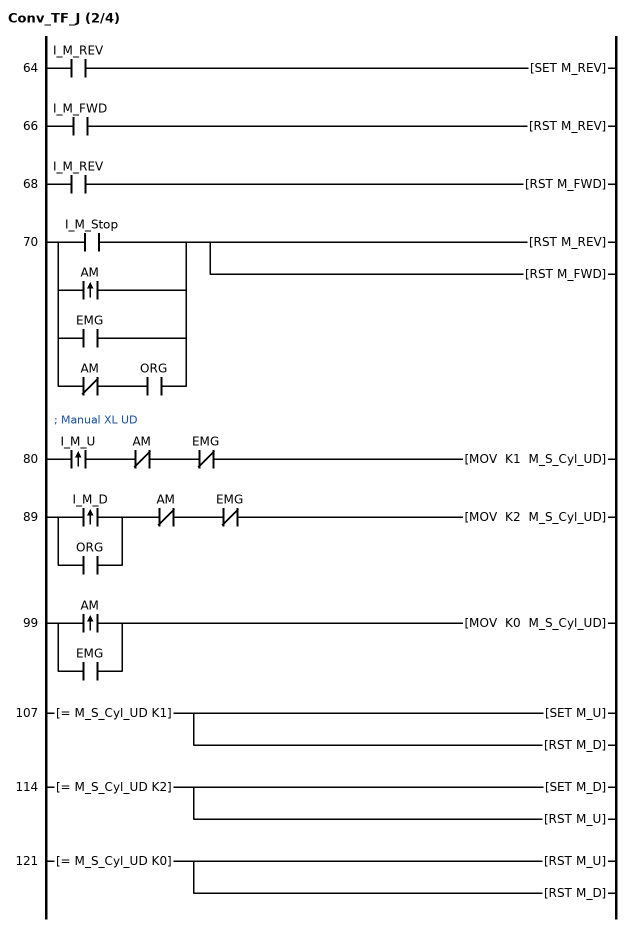
[picture p24: ladder of Conv_TF_J, rungs at steps 64 to 121]
64    LD      I_M_REV
      SET     M_REV
66    LD      I_M_FWD
      RST     M_REV
68    LD      I_M_REV
      RST     M_FWD
70    LD      I_M_Stop
      ORP     AM
      OR      EMG
      LDI     AM
      AND     ORG
      ORB
      RST     M_REV
      RST     M_FWD
; Manual XL UD
80    LDP     I_M_U
      ANI     AM
      ANI     EMG
      MOV     K1 M_S_Cyl_UD
89    LDP     I_M_D
      OR      ORG
      ANI     AM
      ANI     EMG
      MOV     K2 M_S_Cyl_UD
99    LDP     AM
      OR      EMG
      MOV     K0 M_S_Cyl_UD
107   LD=     M_S_Cyl_UD K1
      SET     M_U
      RST     M_D
114   LD=     M_S_Cyl_UD K2
      SET     M_D
      RST     M_U
121   LD=     M_S_Cyl_UD K0
      RST     M_U
      RST     M_D
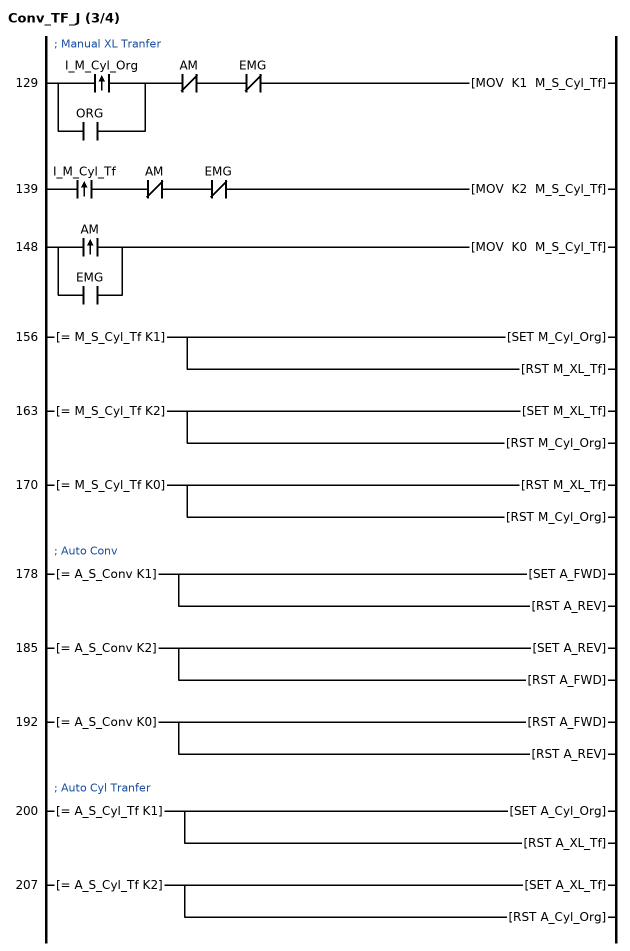
; Manual XL Tranfer
129   LDP     I_M_Cyl_Org
      OR      ORG
      ANI     AM
      ANI     EMG
      MOV     K1 M_S_Cyl_Tf
139   LDP     I_M_Cyl_Tf
      ANI     AM
      ANI     EMG
      MOV     K2 M_S_Cyl_Tf
148   LDP     AM
      OR      EMG
      MOV     K0 M_S_Cyl_Tf
156   LD=     M_S_Cyl_Tf K1
      SET     M_Cyl_Org
      RST     M_XL_Tf
163   LD=     M_S_Cyl_Tf K2
      SET     M_XL_Tf
      RST     M_Cyl_Org
170   LD=     M_S_Cyl_Tf K0
      RST     M_XL_Tf
      RST     M_Cyl_Org
; Auto Conv
178   LD=     A_S_Conv K1
      SET     A_FWD
      RST     A_REV
185   LD=     A_S_Conv K2
      SET     A_REV
      RST     A_FWD
192   LD=     A_S_Conv K0
      RST     A_FWD
      RST     A_REV
; Auto Cyl Tranfer
200   LD=     A_S_Cyl_Tf K1
      SET     A_Cyl_Org
      RST     A_XL_Tf
207   LD=     A_S_Cyl_Tf K2
      SET     A_XL_Tf
      RST     A_Cyl_Org
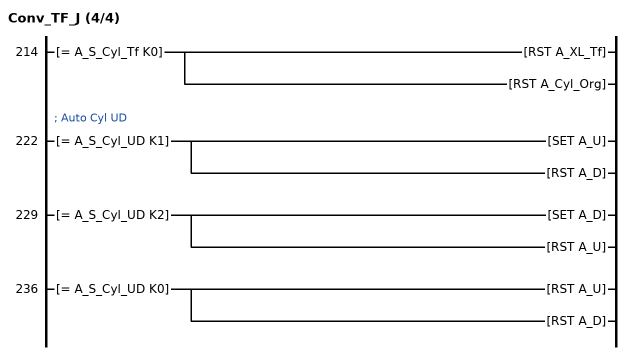
214   LD=     A_S_Cyl_Tf K0
      RST     A_XL_Tf
      RST     A_Cyl_Org
; Auto Cyl UD
222   LD=     A_S_Cyl_UD K1
      SET     A_U
      RST     A_D
229   LD=     A_S_Cyl_UD K2
      SET     A_D
      RST     A_U
236   LD=     A_S_Cyl_UD K0
      RST     A_U
      RST     A_D
END_FUNCTION_BLOCK

FUNCTION_BLOCK Conv_Wait
VAR_INPUT
  AM : BOOL;
  EMG : BOOL;
END_VAR
VAR_OUTPUT
  FWD : BOOL;
  Stopper_Up : BOOL;
  Stopper_Down : BOOL;
END_VAR
VAR
  M_FWD : BOOL;
  M_U : BOOL;
  A_U : BOOL;
  M_D : BOOL;
  A_D : BOOL;
  M_S_Stp : INT;
END_VAR
VAR_INPUT
  I_M_FWD : BOOL;
  I_M_Stop : BOOL;
  I_M_U : BOOL;
  I_M_D : BOOL;
  A_FWD : BOOL;
  A_S_Stp : INT;
  L_C : BOOL;
  ORG : BOOL;
END_VAR
VAR_OUTPUT
  S_Org : BOOL;
END_VAR
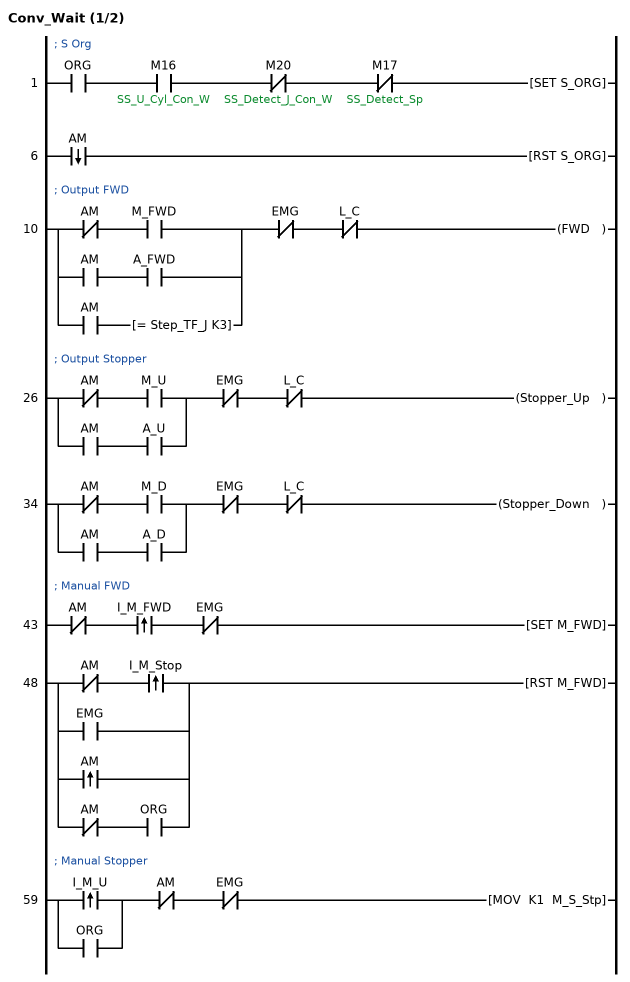
; S Org
1     LD      ORG
      AND     M16  ; SS_U_Cyl_Con_W
      ANI     M20  ; SS_Detect_J_Con_W
      ANI     M17  ; SS_Detect_Sp
      SET     S_ORG
6     LDF     AM
      RST     S_ORG
; Output FWD
10    LDI     AM
      AND     M_FWD
      LD      AM
      AND     A_FWD
      ORB
      LD      AM
      AND=    Step_TF_J K3
      ORB
      ANI     EMG
      ANI     L_C
      OUT     FWD
; Output Stopper
26    LDI     AM
      AND     M_U
      LD      AM
      AND     A_U
      ORB
      ANI     EMG
      ANI     L_C
      OUT     Stopper_Up
34    LDI     AM
      AND     M_D
      LD      AM
      AND     A_D
      ORB
      ANI     EMG
      ANI     L_C
      OUT     Stopper_Down
; Manual FWD
43    LDI     AM
      ANDP    I_M_FWD
      ANI     EMG
      SET     M_FWD
48    LDI     AM
      ANDP    I_M_Stop
      OR      EMG
      ORP     AM
      LDI     AM
      AND     ORG
      ORB
      RST     M_FWD
; Manual Stopper
59    LDP     I_M_U
      OR      ORG
      ANI     AM
      ANI     EMG
      MOV     K1 M_S_Stp
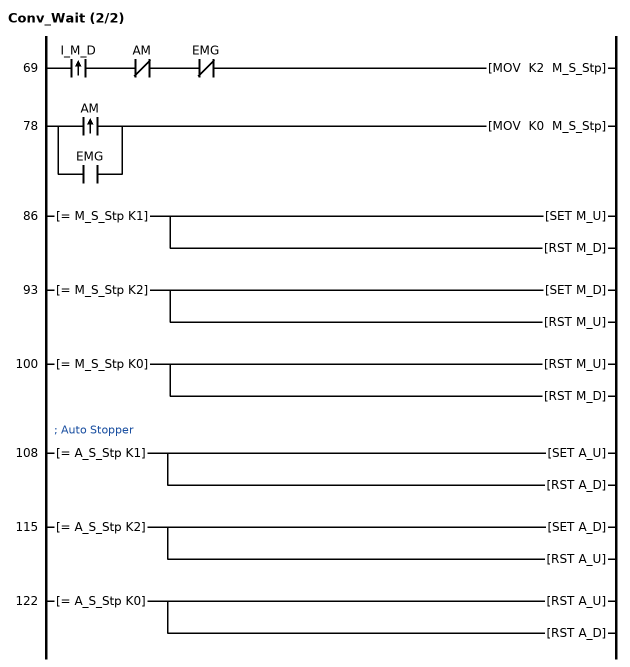
69    LDP     I_M_D
      ANI     AM
      ANI     EMG
      MOV     K2 M_S_Stp
78    LDP     AM
      OR      EMG
      MOV     K0 M_S_Stp
86    LD=     M_S_Stp K1
      SET     M_U
      RST     M_D
93    LD=     M_S_Stp K2
      SET     M_D
      RST     M_U
100   LD=     M_S_Stp K0
      RST     M_U
      RST     M_D
; Auto Stopper
108   LD=     A_S_Stp K1
      SET     A_U
      RST     A_D
115   LD=     A_S_Stp K2
      SET     A_D
      RST     A_U
122   LD=     A_S_Stp K0
      RST     A_U
      RST     A_D
END_FUNCTION_BLOCK

FUNCTION_BLOCK C_Cyl_TF_J
VAR_INPUT
  AM : BOOL;
  EMG : BOOL;
END_VAR
VAR
  M_U : BOOL;
  A_U : BOOL;
  M_D : BOOL;
  A_D : BOOL;
  M_S_Cyl_UD : INT;
  M_Org_XL_Tf : BOOL;
  A_Org_XL_Tf : BOOL;
  M_Tf_XL_Tf : BOOL;
  A_Tf_XL_Tf : BOOL;
END_VAR
VAR_INPUT
  I_M_U : BOOL;
  I_M_D : BOOL;
  I_M_Sol_Org : BOOL;
  I_M_Sol_Tf : BOOL;
  A_Status_XL_U : INT;
END_VAR
VAR
  M_Status_XL_Tf : INT;
END_VAR
VAR_INPUT
  A_S_Cyl_Tf : INT;
  ORG : BOOL;
END_VAR
VAR_OUTPUT
  XL_U : BOOL;
  XL_D : BOOL;
  Sol_Org : BOOL;
  Sol_Tranfer : BOOL;
  S_Org : BOOL;
END_VAR
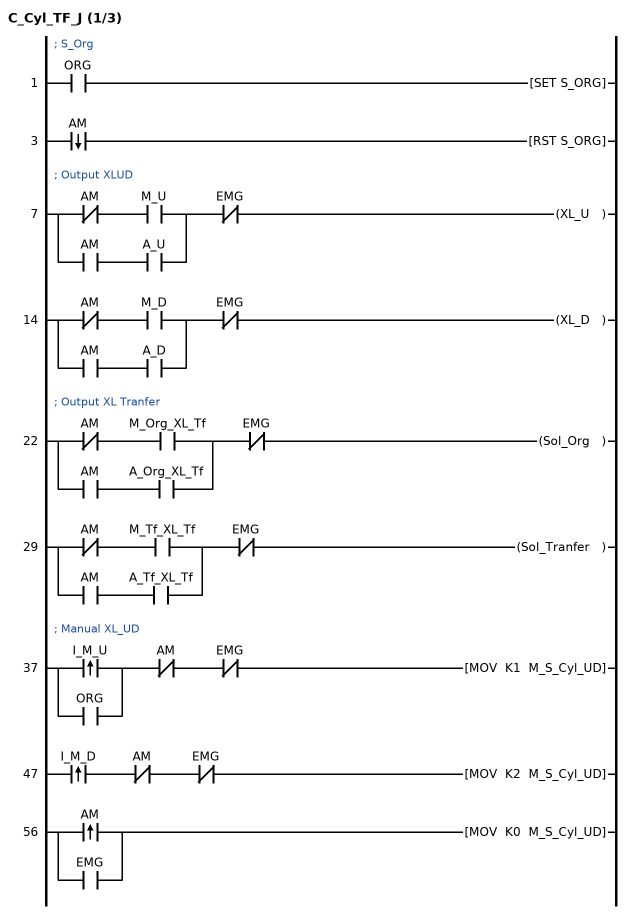
; S_Org
1     LD      ORG
      SET     S_ORG
3     LDF     AM
      RST     S_ORG
; Output XLUD
7     LDI     AM
      AND     M_U
      LD      AM
      AND     A_U
      ORB
      ANI     EMG
      OUT     XL_U
14    LDI     AM
      AND     M_D
      LD      AM
      AND     A_D
      ORB
      ANI     EMG
      OUT     XL_D
; Output XL Tranfer
22    LDI     AM
      AND     M_Org_XL_Tf
      LD      AM
      AND     A_Org_XL_Tf
      ORB
      ANI     EMG
      OUT     Sol_Org
29    LDI     AM
      AND     M_Tf_XL_Tf
      LD      AM
      AND     A_Tf_XL_Tf
      ORB
      ANI     EMG
      OUT     Sol_Tranfer
; Manual XL_UD
37    LDP     I_M_U
      OR      ORG
      ANI     AM
      ANI     EMG
      MOV     K1 M_S_Cyl_UD
47    LDP     I_M_D
      ANI     AM
      ANI     EMG
      MOV     K2 M_S_Cyl_UD
56    LDP     AM
      OR      EMG
      MOV     K0 M_S_Cyl_UD
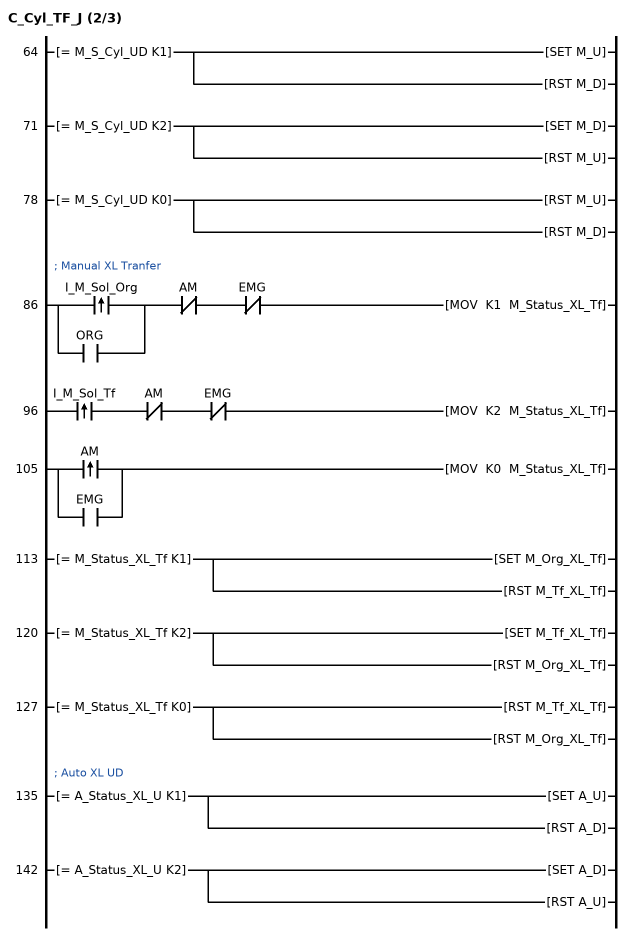
64    LD=     M_S_Cyl_UD K1
      SET     M_U
      RST     M_D
71    LD=     M_S_Cyl_UD K2
      SET     M_D
      RST     M_U
78    LD=     M_S_Cyl_UD K0
      RST     M_U
      RST     M_D
; Manual XL Tranfer
86    LDP     I_M_Sol_Org
      OR      ORG
      ANI     AM
      ANI     EMG
      MOV     K1 M_Status_XL_Tf
96    LDP     I_M_Sol_Tf
      ANI     AM
      ANI     EMG
      MOV     K2 M_Status_XL_Tf
105   LDP     AM
      OR      EMG
      MOV     K0 M_Status_XL_Tf
113   LD=     M_Status_XL_Tf K1
      SET     M_Org_XL_Tf
      RST     M_Tf_XL_Tf
120   LD=     M_Status_XL_Tf K2
      SET     M_Tf_XL_Tf
      RST     M_Org_XL_Tf
127   LD=     M_Status_XL_Tf K0
      RST     M_Tf_XL_Tf
      RST     M_Org_XL_Tf
; Auto XL UD
135   LD=     A_Status_XL_U K1
      SET     A_U
      RST     A_D
142   LD=     A_Status_XL_U K2
      SET     A_D
      RST     A_U
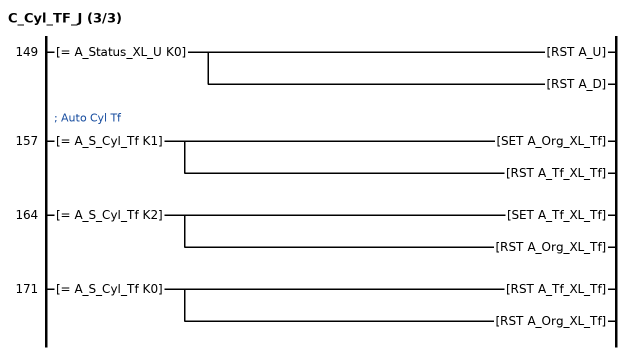
149   LD=     A_Status_XL_U K0
      RST     A_U
      RST     A_D
; Auto Cyl Tf
157   LD=     A_S_Cyl_Tf K1
      SET     A_Org_XL_Tf
      RST     A_Tf_XL_Tf
164   LD=     A_S_Cyl_Tf K2
      SET     A_Tf_XL_Tf
      RST     A_Org_XL_Tf
171   LD=     A_S_Cyl_Tf K0
      RST     A_Tf_XL_Tf
      RST     A_Org_XL_Tf
END_FUNCTION_BLOCK

FUNCTION_BLOCK C_Cyl_TF_SP
VAR_INPUT
  AM : BOOL;
  EMG : BOOL;
  I_M_U : BOOL;
  I_M_D : BOOL;
  I_M_Sol_Org : BOOL;
  I_M_Sol_Tf : BOOL;
  I_M_XL_Kep_SP1 : BOOL;
  I_M_XL_Nha_SP1 : BOOL;
END_VAR
VAR
  Step_Run : INT;
  Flag_Run : BOOL;
  Full_XL_Ready : BOOL;
  Delay_Kep_Sp : TIMER;
END_VAR
VAR_INPUT
  I_M_XL_Kep_SP2 : BOOL;
  I_M_XL_Nha_SP2 : BOOL;
  A_Status_XL_U : INT;
  A_S_Cyl_Tf : INT;
  A_S_Cyl_Kep_1 : INT;
  A_S_Cyl_Kep_2 : INT;
  ORG : BOOL;
END_VAR
VAR_OUTPUT
  XL_U : BOOL;
  XL_D : BOOL;
  Sol_Org : BOOL;
  Sol_Tranfer : BOOL;
  XL_Kep_SP1 : BOOL;
  XL_Mo_SP1 : BOOL;
  XL_Kep_SP2 : BOOL;
  XL_Mo_SP2 : BOOL;
END_VAR
VAR
  M_U : BOOL;
  A_U : BOOL;
  M_D : BOOL;
  A_D : BOOL;
  M_S_Cyl_UD : INT;
  M_Org_XL_Tf : BOOL;
  A_Org_XL_Tf : BOOL;
  M_Tf_XL_Tf : BOOL;
  A_Tf_XL_Tf : BOOL;
  M_Status_XL_Tf : INT;
  M_Kep_SP1 : BOOL;
  A_Kep_SP1 : BOOL;
  M_Nha_SP1 : BOOL;
  A_Nha_SP1 : BOOL;
  M_Status_XL_Kep_Sp1 : INT;
  M_Kep_SP2 : BOOL;
  A_Kep_SP2 : BOOL;
  M_Nha_SP2 : BOOL;
  A_Nha_SP2 : BOOL;
  M_Status_XL_Kep_Sp2 : INT;
END_VAR
VAR_OUTPUT
  S_ORG : BOOL;
END_VAR
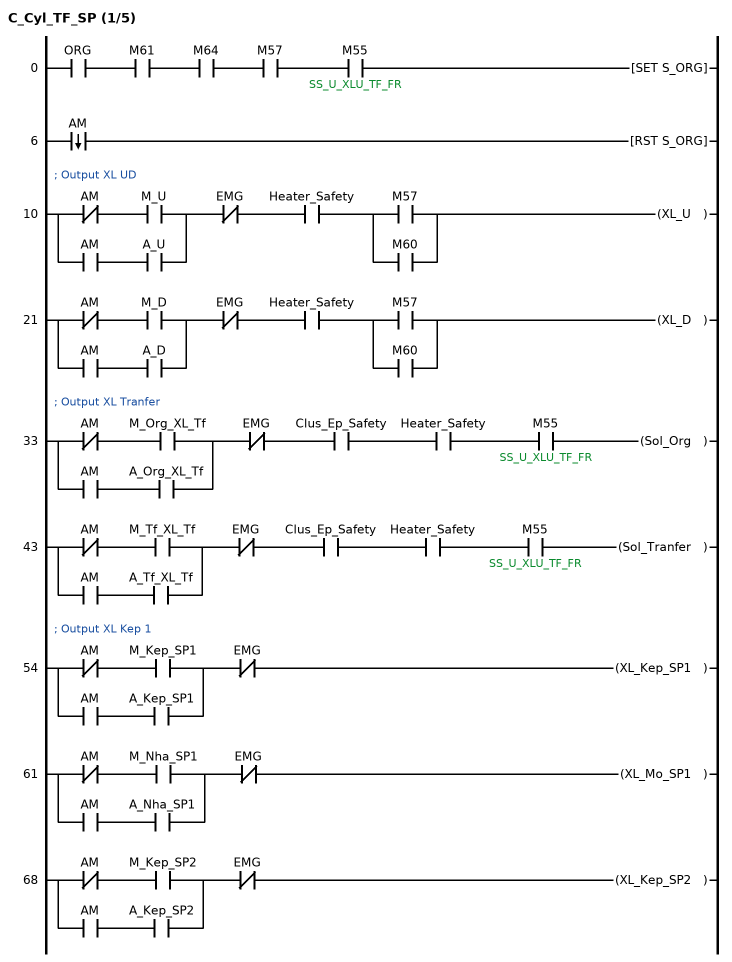
0     LD      ORG
      AND     M61
      AND     M64
      AND     M57
      AND     M55  ; SS_U_XLU_TF_FR
      SET     S_ORG
6     LDF     AM
      RST     S_ORG
; Output XL UD
10    LDI     AM
      AND     M_U
      LD      AM
      AND     A_U
      ORB
      ANI     EMG
      AND     Heater_Safety
      LD      M57
      OR      M60
      ANB
      OUT     XL_U
21    LDI     AM
      AND     M_D
      LD      AM
      AND     A_D
      ORB
      ANI     EMG
      AND     Heater_Safety
      LD      M57
      OR      M60
      ANB
      OUT     XL_D
; Output XL Tranfer
33    LDI     AM
      AND     M_Org_XL_Tf
      LD      AM
      AND     A_Org_XL_Tf
      ORB
      ANI     EMG
      AND     Clus_Ep_Safety
      AND     Heater_Safety
      AND     M55  ; SS_U_XLU_TF_FR
      OUT     Sol_Org
43    LDI     AM
      AND     M_Tf_XL_Tf
      LD      AM
      AND     A_Tf_XL_Tf
      ORB
      ANI     EMG
      AND     Clus_Ep_Safety
      AND     Heater_Safety
      AND     M55  ; SS_U_XLU_TF_FR
      OUT     Sol_Tranfer
; Output XL Kep 1
54    LDI     AM
      AND     M_Kep_SP1
      LD      AM
      AND     A_Kep_SP1
      ORB
      ANI     EMG
      OUT     XL_Kep_SP1
61    LDI     AM
      AND     M_Nha_SP1
      LD      AM
      AND     A_Nha_SP1
      ORB
      ANI     EMG
      OUT     XL_Mo_SP1
68    LDI     AM
      AND     M_Kep_SP2
      LD      AM
      AND     A_Kep_SP2
      ORB
      ANI     EMG
      OUT     XL_Kep_SP2
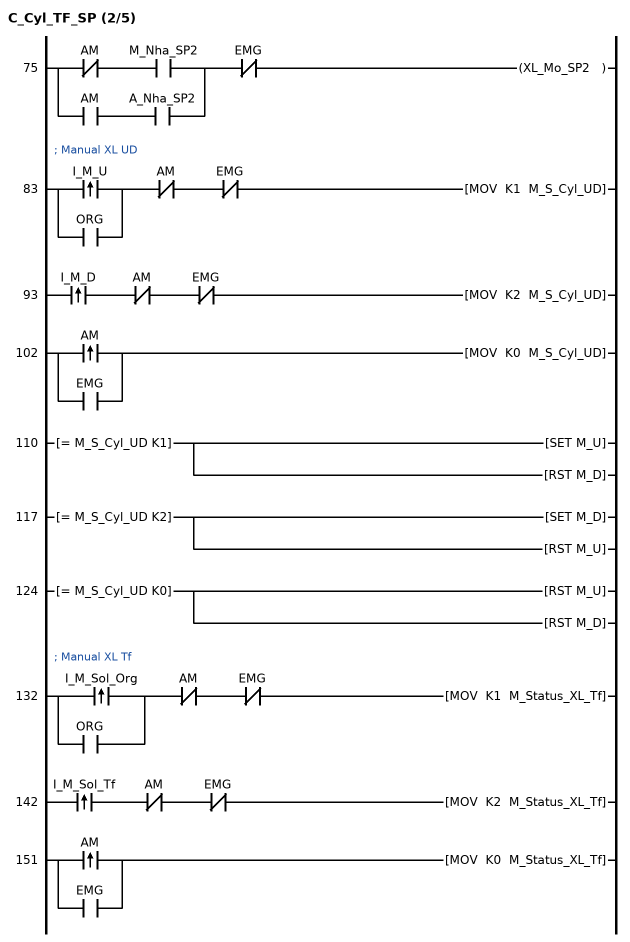
75    LDI     AM
      AND     M_Nha_SP2
      LD      AM
      AND     A_Nha_SP2
      ORB
      ANI     EMG
      OUT     XL_Mo_SP2
; Manual XL UD
83    LDP     I_M_U
      OR      ORG
      ANI     AM
      ANI     EMG
      MOV     K1 M_S_Cyl_UD
93    LDP     I_M_D
      ANI     AM
      ANI     EMG
      MOV     K2 M_S_Cyl_UD
102   LDP     AM
      OR      EMG
      MOV     K0 M_S_Cyl_UD
110   LD=     M_S_Cyl_UD K1
      SET     M_U
      RST     M_D
117   LD=     M_S_Cyl_UD K2
      SET     M_D
      RST     M_U
124   LD=     M_S_Cyl_UD K0
      RST     M_U
      RST     M_D
; Manual XL Tf
132   LDP     I_M_Sol_Org
      OR      ORG
      ANI     AM
      ANI     EMG
      MOV     K1 M_Status_XL_Tf
142   LDP     I_M_Sol_Tf
      ANI     AM
      ANI     EMG
      MOV     K2 M_Status_XL_Tf
151   LDP     AM
      OR      EMG
      MOV     K0 M_Status_XL_Tf
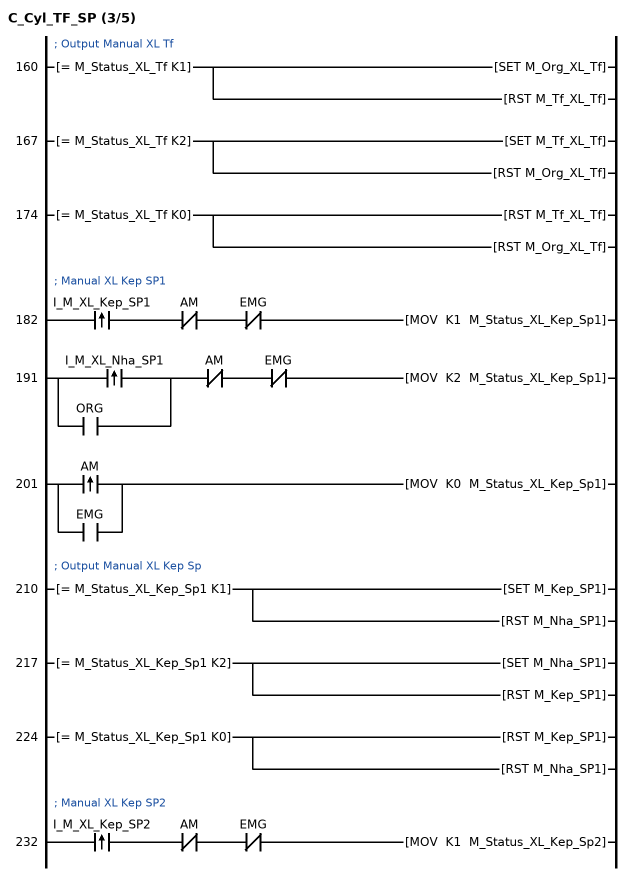
; Output Manual XL Tf
160   LD=     M_Status_XL_Tf K1
      SET     M_Org_XL_Tf
      RST     M_Tf_XL_Tf
167   LD=     M_Status_XL_Tf K2
      SET     M_Tf_XL_Tf
      RST     M_Org_XL_Tf
174   LD=     M_Status_XL_Tf K0
      RST     M_Tf_XL_Tf
      RST     M_Org_XL_Tf
; Manual XL Kep SP1
182   LDP     I_M_XL_Kep_SP1
      ANI     AM
      ANI     EMG
      MOV     K1 M_Status_XL_Kep_Sp1
191   LDP     I_M_XL_Nha_SP1
      OR      ORG
      ANI     AM
      ANI     EMG
      MOV     K2 M_Status_XL_Kep_Sp1
201   LDP     AM
      OR      EMG
      MOV     K0 M_Status_XL_Kep_Sp1
; Output Manual XL Kep Sp
210   LD=     M_Status_XL_Kep_Sp1 K1
      SET     M_Kep_SP1
      RST     M_Nha_SP1
217   LD=     M_Status_XL_Kep_Sp1 K2
      SET     M_Nha_SP1
      RST     M_Kep_SP1
224   LD=     M_Status_XL_Kep_Sp1 K0
      RST     M_Kep_SP1
      RST     M_Nha_SP1
; Manual XL Kep SP2
232   LDP     I_M_XL_Kep_SP2
      ANI     AM
      ANI     EMG
      MOV     K1 M_Status_XL_Kep_Sp2
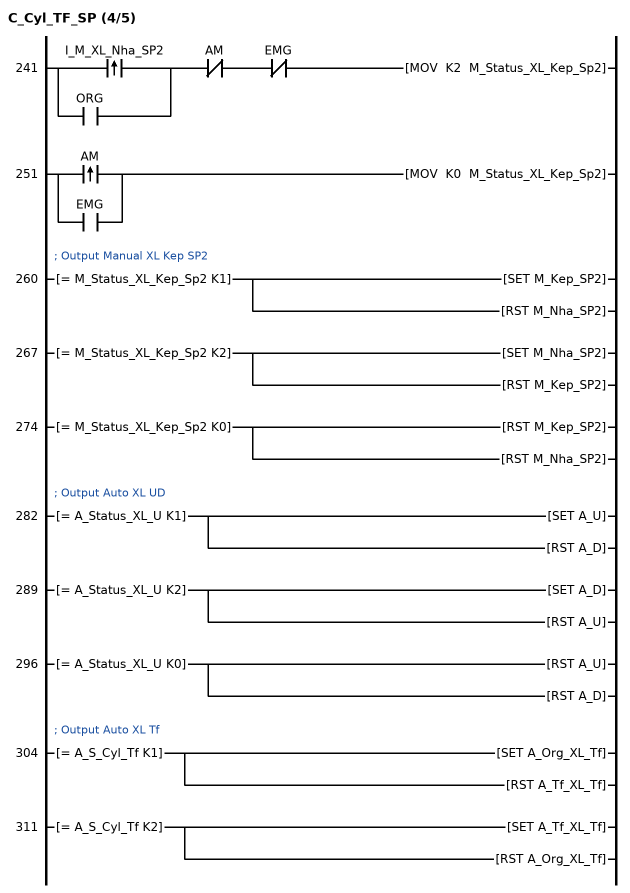
241   LDP     I_M_XL_Nha_SP2
      OR      ORG
      ANI     AM
      ANI     EMG
      MOV     K2 M_Status_XL_Kep_Sp2
251   LDP     AM
      OR      EMG
      MOV     K0 M_Status_XL_Kep_Sp2
; Output Manual XL Kep SP2
260   LD=     M_Status_XL_Kep_Sp2 K1
      SET     M_Kep_SP2
      RST     M_Nha_SP2
267   LD=     M_Status_XL_Kep_Sp2 K2
      SET     M_Nha_SP2
      RST     M_Kep_SP2
274   LD=     M_Status_XL_Kep_Sp2 K0
      RST     M_Kep_SP2
      RST     M_Nha_SP2
; Output Auto XL UD
282   LD=     A_Status_XL_U K1
      SET     A_U
      RST     A_D
289   LD=     A_Status_XL_U K2
      SET     A_D
      RST     A_U
296   LD=     A_Status_XL_U K0
      RST     A_U
      RST     A_D
; Output Auto XL Tf
304   LD=     A_S_Cyl_Tf K1
      SET     A_Org_XL_Tf
      RST     A_Tf_XL_Tf
311   LD=     A_S_Cyl_Tf K2
      SET     A_Tf_XL_Tf
      RST     A_Org_XL_Tf
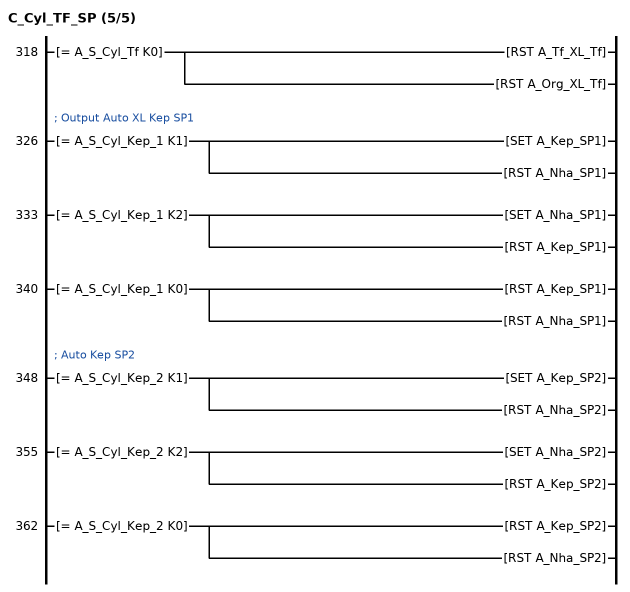
318   LD=     A_S_Cyl_Tf K0
      RST     A_Tf_XL_Tf
      RST     A_Org_XL_Tf
; Output Auto XL Kep SP1
326   LD=     A_S_Cyl_Kep_1 K1
      SET     A_Kep_SP1
      RST     A_Nha_SP1
333   LD=     A_S_Cyl_Kep_1 K2
      SET     A_Nha_SP1
      RST     A_Kep_SP1
340   LD=     A_S_Cyl_Kep_1 K0
      RST     A_Kep_SP1
      RST     A_Nha_SP1
; Auto Kep SP2
348   LD=     A_S_Cyl_Kep_2 K1
      SET     A_Kep_SP2
      RST     A_Nha_SP2
355   LD=     A_S_Cyl_Kep_2 K2
      SET     A_Nha_SP2
      RST     A_Kep_SP2
362   LD=     A_S_Cyl_Kep_2 K0
      RST     A_Kep_SP2
      RST     A_Nha_SP2
END_FUNCTION_BLOCK

FUNCTION_BLOCK Conv_Out
VAR_INPUT
  AM : BOOL;
  EMG : BOOL;
END_VAR
VAR_OUTPUT
  R_FWD : BOOL;
  Stopper_Up : BOOL;
  Stopper_Down : BOOL;
  Cyl_U_Jig : BOOL;
  Cyl_D_Jig : BOOL;
END_VAR
VAR_INPUT
  I_M_U_S : BOOL;
  I_M_D_S : BOOL;
  I_M_U_Jig : BOOL;
  I_M_D_Jig : BOOL;
  I_M_FWD : BOOL;
  I_M_Stop : BOOL;
END_VAR
VAR
  M_FWD : BOOL;
  M_U_Jig : BOOL;
  A_U_Jig : BOOL;
  M_S_Cyl_UD : INT;
  M_D_Jig : BOOL;
  A_D_Jig : BOOL;
  M_U_S : BOOL;
  A_U_S : BOOL;
  M_D_S : BOOL;
  A_D_S : BOOL;
  M_S_Stp : INT;
END_VAR
VAR_INPUT
  ORG : BOOL;
END_VAR
VAR_OUTPUT
  S_Org : BOOL;
  Sol_Do1 : BOOL;
  Sol_Do2 : BOOL;
END_VAR
VAR_INPUT
  A_S_Cyl_UD : INT;
  A_S_Stp : INT;
  A_FWD : BOOL;
  I_M_Do1 : BOOL;
  I_M_Do2 : BOOL;
  A_S_Do : INT;
END_VAR
VAR
  M_Do1 : BOOL;
  A_Do1 : BOOL;
  M_Do2 : BOOL;
  A_Do2 : BOOL;
  M_S_Do : INT;
END_VAR
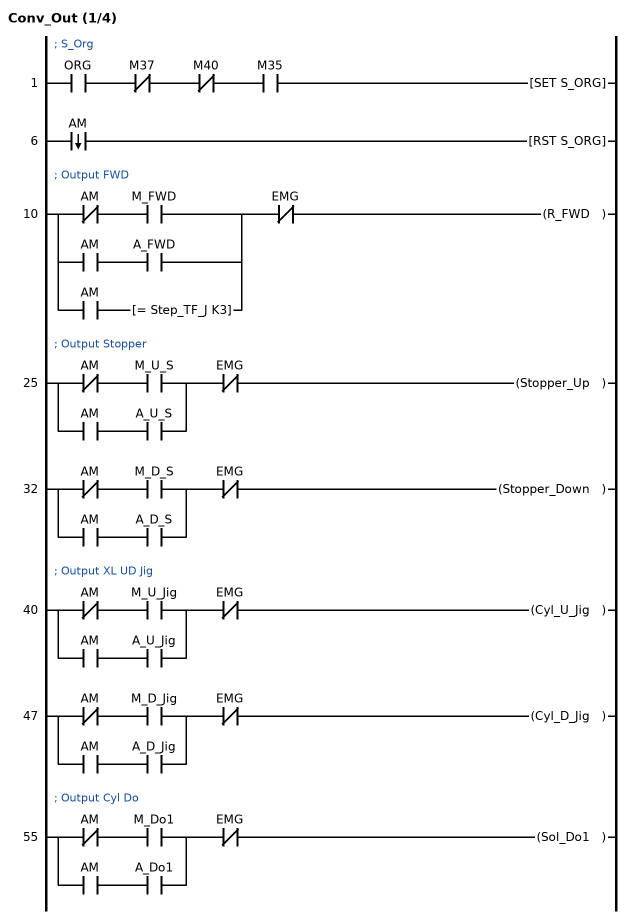
; S_Org
1     LD      ORG
      ANI     M37
      ANI     M40
      AND     M35
      SET     S_ORG
6     LDF     AM
      RST     S_ORG
; Output FWD
10    LDI     AM
      AND     M_FWD
      LD      AM
      AND     A_FWD
      ORB
      LD      AM
      AND=    Step_TF_J K3
      ORB
      ANI     EMG
      OUT     R_FWD
; Output Stopper
25    LDI     AM
      AND     M_U_S
      LD      AM
      AND     A_U_S
      ORB
      ANI     EMG
      OUT     Stopper_Up
32    LDI     AM
      AND     M_D_S
      LD      AM
      AND     A_D_S
      ORB
      ANI     EMG
      OUT     Stopper_Down
; Output XL UD Jig
40    LDI     AM
      AND     M_U_Jig
      LD      AM
      AND     A_U_Jig
      ORB
      ANI     EMG
      OUT     Cyl_U_Jig
47    LDI     AM
      AND     M_D_Jig
      LD      AM
      AND     A_D_Jig
      ORB
      ANI     EMG
      OUT     Cyl_D_Jig
; Output Cyl Do
55    LDI     AM
      AND     M_Do1
      LD      AM
      AND     A_Do1
      ORB
      ANI     EMG
      OUT     Sol_Do1
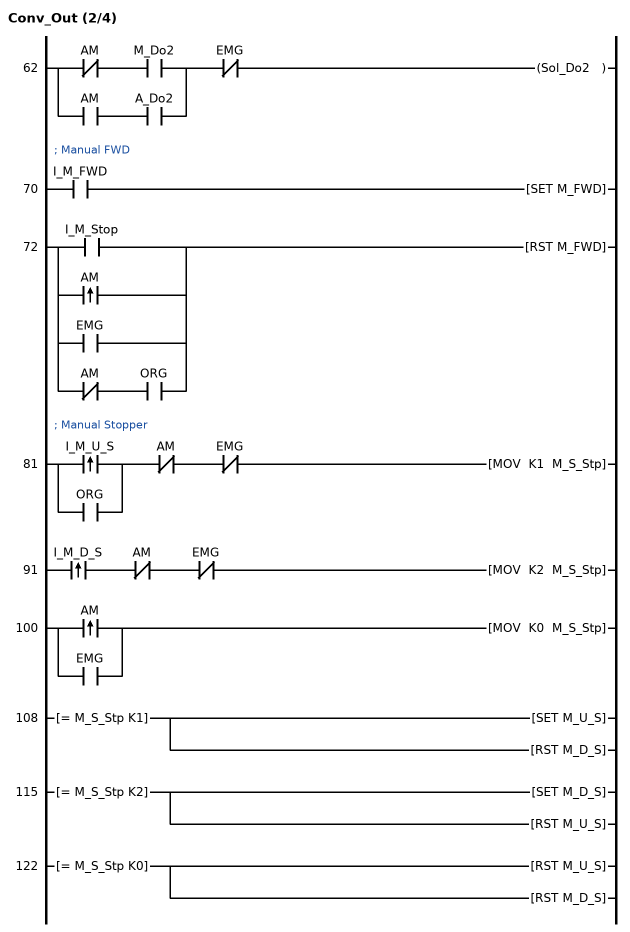
62    LDI     AM
      AND     M_Do2
      LD      AM
      AND     A_Do2
      ORB
      ANI     EMG
      OUT     Sol_Do2
; Manual FWD
70    LD      I_M_FWD
      SET     M_FWD
72    LD      I_M_Stop
      ORP     AM
      OR      EMG
      LDI     AM
      AND     ORG
      ORB
      RST     M_FWD
; Manual Stopper
81    LDP     I_M_U_S
      OR      ORG
      ANI     AM
      ANI     EMG
      MOV     K1 M_S_Stp
91    LDP     I_M_D_S
      ANI     AM
      ANI     EMG
      MOV     K2 M_S_Stp
100   LDP     AM
      OR      EMG
      MOV     K0 M_S_Stp
108   LD=     M_S_Stp K1
      SET     M_U_S
      RST     M_D_S
115   LD=     M_S_Stp K2
      SET     M_D_S
      RST     M_U_S
122   LD=     M_S_Stp K0
      RST     M_U_S
      RST     M_D_S
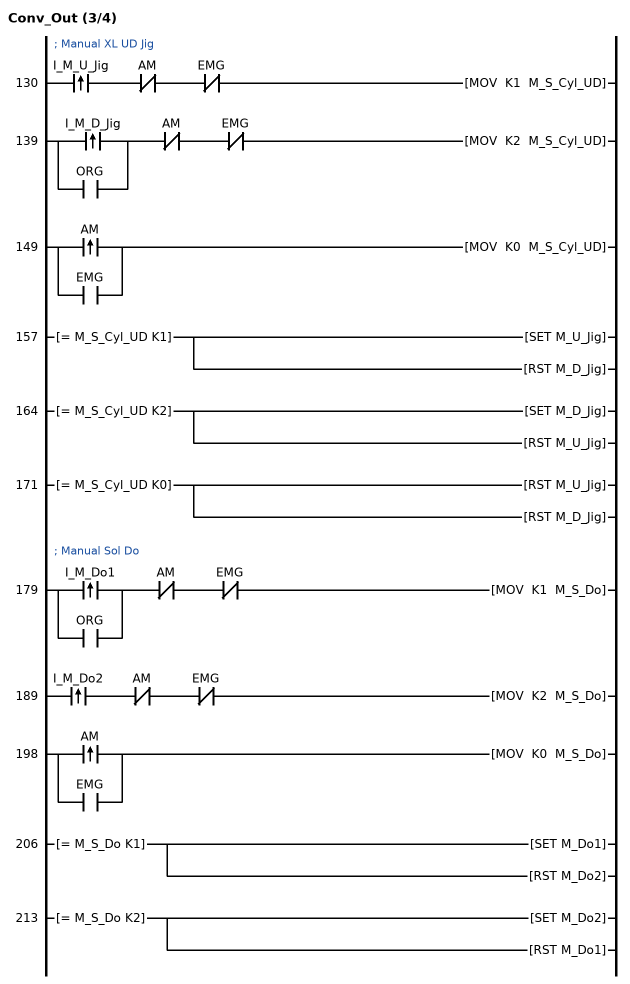
; Manual XL UD Jig
130   LDP     I_M_U_Jig
      ANI     AM
      ANI     EMG
      MOV     K1 M_S_Cyl_UD
139   LDP     I_M_D_Jig
      OR      ORG
      ANI     AM
      ANI     EMG
      MOV     K2 M_S_Cyl_UD
149   LDP     AM
      OR      EMG
      MOV     K0 M_S_Cyl_UD
157   LD=     M_S_Cyl_UD K1
      SET     M_U_Jig
      RST     M_D_Jig
164   LD=     M_S_Cyl_UD K2
      SET     M_D_Jig
      RST     M_U_Jig
171   LD=     M_S_Cyl_UD K0
      RST     M_U_Jig
      RST     M_D_Jig
; Manual Sol Do
179   LDP     I_M_Do1
      OR      ORG
      ANI     AM
      ANI     EMG
      MOV     K1 M_S_Do
189   LDP     I_M_Do2
      ANI     AM
      ANI     EMG
      MOV     K2 M_S_Do
198   LDP     AM
      OR      EMG
      MOV     K0 M_S_Do
206   LD=     M_S_Do K1
      SET     M_Do1
      RST     M_Do2
213   LD=     M_S_Do K2
      SET     M_Do2
      RST     M_Do1
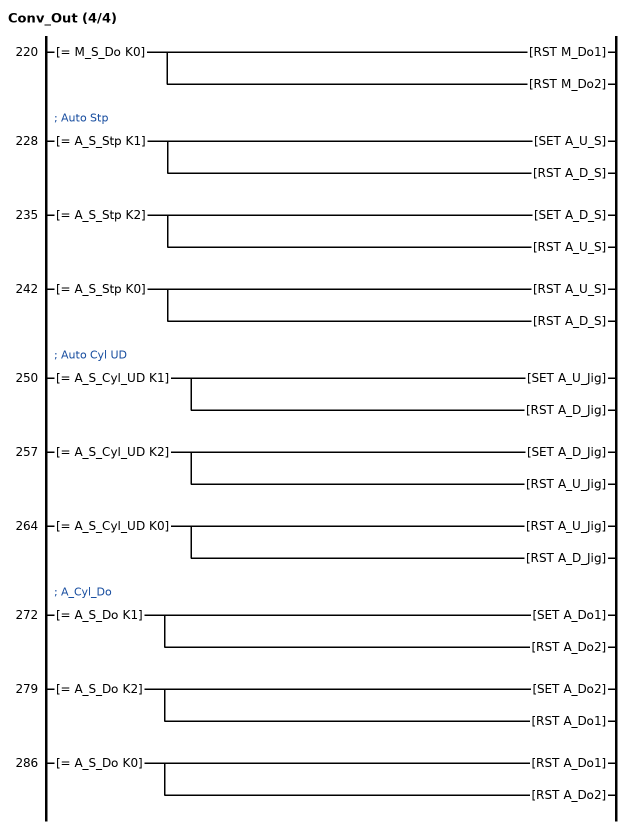
220   LD=     M_S_Do K0
      RST     M_Do1
      RST     M_Do2
; Auto Stp
228   LD=     A_S_Stp K1
      SET     A_U_S
      RST     A_D_S
235   LD=     A_S_Stp K2
      SET     A_D_S
      RST     A_U_S
242   LD=     A_S_Stp K0
      RST     A_U_S
      RST     A_D_S
; Auto Cyl UD
250   LD=     A_S_Cyl_UD K1
      SET     A_U_Jig
      RST     A_D_Jig
257   LD=     A_S_Cyl_UD K2
      SET     A_D_Jig
      RST     A_U_Jig
264   LD=     A_S_Cyl_UD K0
      RST     A_U_Jig
      RST     A_D_Jig
; A_Cyl_Do
272   LD=     A_S_Do K1
      SET     A_Do1
      RST     A_Do2
279   LD=     A_S_Do K2
      SET     A_Do2
      RST     A_Do1
286   LD=     A_S_Do K0
      RST     A_Do1
      RST     A_Do2
END_FUNCTION_BLOCK

FUNCTION_BLOCK Heater
VAR_INPUT
  AM : BOOL;
  EMG : BOOL;
END_VAR
VAR_OUTPUT
  ON_Heater : BOOL;
  XL_U : BOOL;
  XL_D : BOOL;
  ON_Center : BOOL;
  OFF_Center : BOOL;
END_VAR
VAR_INPUT
  I_M_U : BOOL;
  I_M_D : BOOL;
  I_M_On_Center : BOOL;
  I_M_Off_Center : BOOL;
END_VAR
VAR
  M_U : BOOL;
  A_U : BOOL;
  M_D : BOOL;
  A_D : BOOL;
  M_S_Cyl_UD : INT;
  M_ON_Center : BOOL;
  A_ON_Center : BOOL;
  M_OFF_Center : BOOL;
  A_OFF_Center : BOOL;
  M_Status_Center : INT;
END_VAR
VAR_INPUT
  I_ON_Heater : BOOL;
  A_ON_Heater : BOOL;
  A_S_Cyl_UD : INT;
  A_Status_Center : INT;
  T_Real : REAL;
  T_Limit : REAL;
  ORG : BOOL;
END_VAR
VAR_OUTPUT
  S_ORG : BOOL;
END_VAR
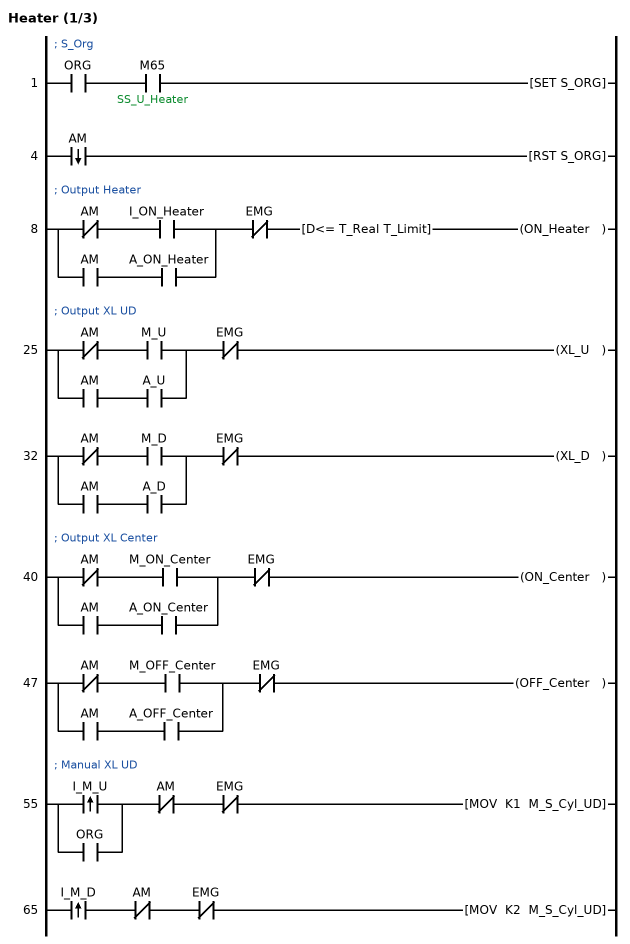
; S_Org
1     LD      ORG
      AND     M65  ; SS_U_Heater
      SET     S_ORG
4     LDF     AM
      RST     S_ORG
; Output Heater
8     LDI     AM
      AND     I_ON_Heater
      LD      AM
      AND     A_ON_Heater
      ORB
      ANI     EMG
      ANDD<=  T_Real T_Limit
      OUT     ON_Heater
; Output XL UD
25    LDI     AM
      AND     M_U
      LD      AM
      AND     A_U
      ORB
      ANI     EMG
      OUT     XL_U
32    LDI     AM
      AND     M_D
      LD      AM
      AND     A_D
      ORB
      ANI     EMG
      OUT     XL_D
; Output XL Center
40    LDI     AM
      AND     M_ON_Center
      LD      AM
      AND     A_ON_Center
      ORB
      ANI     EMG
      OUT     ON_Center
47    LDI     AM
      AND     M_OFF_Center
      LD      AM
      AND     A_OFF_Center
      ORB
      ANI     EMG
      OUT     OFF_Center
; Manual XL UD
55    LDP     I_M_U
      OR      ORG
      ANI     AM
      ANI     EMG
      MOV     K1 M_S_Cyl_UD
65    LDP     I_M_D
      ANI     AM
      ANI     EMG
      MOV     K2 M_S_Cyl_UD
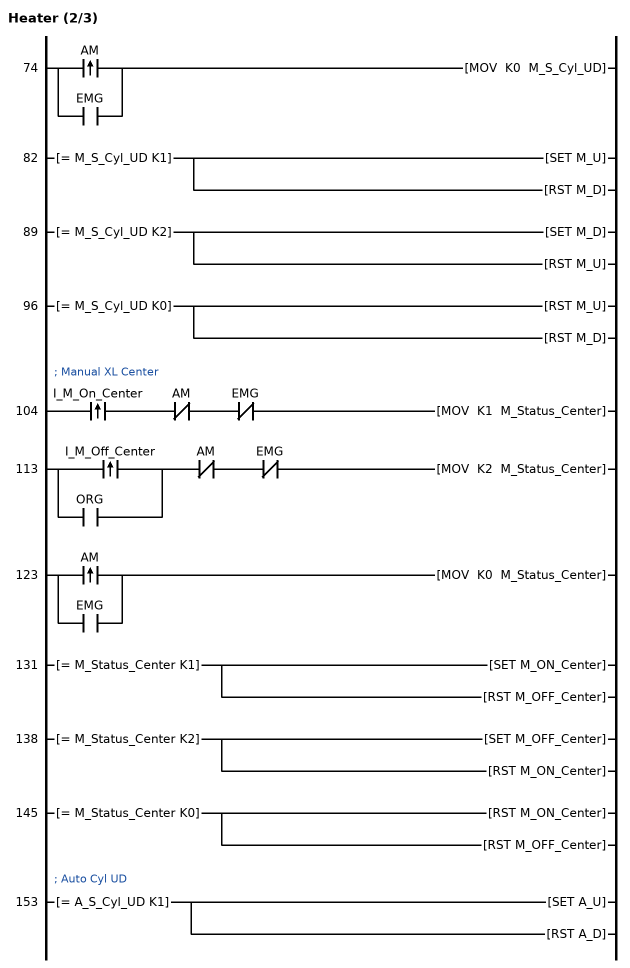
74    LDP     AM
      OR      EMG
      MOV     K0 M_S_Cyl_UD
82    LD=     M_S_Cyl_UD K1
      SET     M_U
      RST     M_D
89    LD=     M_S_Cyl_UD K2
      SET     M_D
      RST     M_U
96    LD=     M_S_Cyl_UD K0
      RST     M_U
      RST     M_D
; Manual XL Center
104   LDP     I_M_On_Center
      ANI     AM
      ANI     EMG
      MOV     K1 M_Status_Center
113   LDP     I_M_Off_Center
      OR      ORG
      ANI     AM
      ANI     EMG
      MOV     K2 M_Status_Center
123   LDP     AM
      OR      EMG
      MOV     K0 M_Status_Center
131   LD=     M_Status_Center K1
      SET     M_ON_Center
      RST     M_OFF_Center
138   LD=     M_Status_Center K2
      SET     M_OFF_Center
      RST     M_ON_Center
145   LD=     M_Status_Center K0
      RST     M_ON_Center
      RST     M_OFF_Center
; Auto Cyl UD
153   LD=     A_S_Cyl_UD K1
      SET     A_U
      RST     A_D
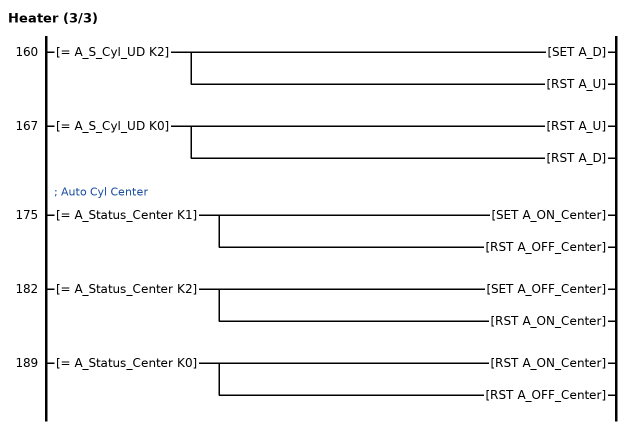
160   LD=     A_S_Cyl_UD K2
      SET     A_D
      RST     A_U
167   LD=     A_S_Cyl_UD K0
      RST     A_U
      RST     A_D
; Auto Cyl Center
175   LD=     A_Status_Center K1
      SET     A_ON_Center
      RST     A_OFF_Center
182   LD=     A_Status_Center K2
      SET     A_OFF_Center
      RST     A_ON_Center
189   LD=     A_Status_Center K0
      RST     A_ON_Center
      RST     A_OFF_Center
END_FUNCTION_BLOCK

FUNCTION_BLOCK Ctr_MC
VAR_INPUT
  I_AM : BOOL;
END_VAR
VAR_OUTPUT
  Flag_Run : BOOL;
  EMG : BOOL;
  AM : BOOL;
  R_Home : BOOL;
END_VAR
VAR_INPUT
  I_RST : BOOL;
  I_ORG : BOOL;
  I_EMG : INT;
END_VAR
VAR
  Delay_R_H : TIMER;
  T_R_H : BOOL;
  T_Auto : TIMER;
END_VAR
VAR_OUTPUT
  Red : BOOL;
  Yel : BOOL;
  Gre : BOOL;
  Buzzer : BOOL;
END_VAR
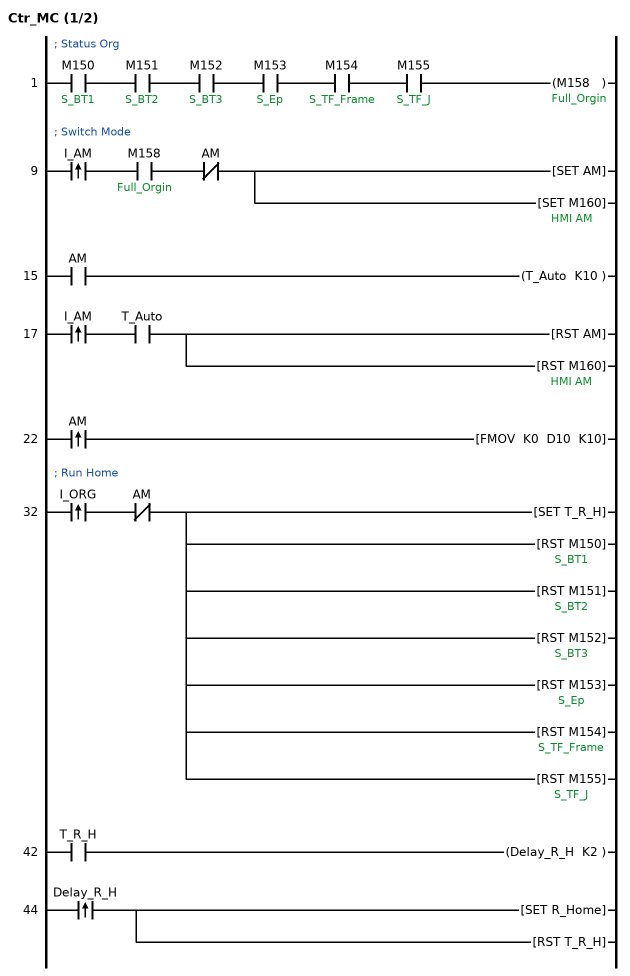
; Status Org
1     LD      M150  ; S_BT1
      AND     M151  ; S_BT2
      AND     M152  ; S_BT3
      AND     M153  ; S_Ep
      AND     M154  ; S_TF_Frame
      AND     M155  ; S_TF_J
      OUT     M158  ; Full_Orgin
; Switch Mode
9     LDP     I_AM
      AND     M158  ; Full_Orgin
      ANI     AM
      SET     AM
      SET     M160  ; HMI AM
15    LD      AM
      OUT     T_Auto K10
17    LDP     I_AM
      AND     T_Auto
      RST     AM
      RST     M160  ; HMI AM
22    LDP     AM
      FMOV    K0 D10 K10
; Run Home
32    LDP     I_ORG
      ANI     AM
      SET     T_R_H
      RST     M150  ; S_BT1
      RST     M151  ; S_BT2
      RST     M152  ; S_BT3
      RST     M153  ; S_Ep
      RST     M154  ; S_TF_Frame
      RST     M155  ; S_TF_J
42    LD      T_R_H
      OUT     Delay_R_H K2
44    LDP     Delay_R_H
      SET     R_Home
      RST     T_R_H
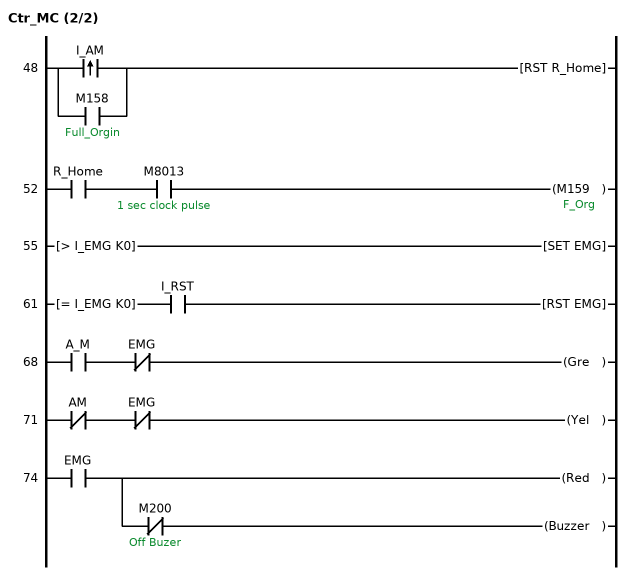
48    LDP     I_AM
      OR      M158  ; Full_Orgin
      RST     R_Home
52    LD      R_Home
      AND     M8013  ; 1 sec clock pulse
      OUT     M159  ; F_Org
55    LD>     I_EMG K0
      SET     EMG
61    LD=     I_EMG K0
      AND     I_RST
      RST     EMG
68    LD      A_M
      ANI     EMG
      OUT     Gre
71    LDI     AM
      ANI     EMG
      OUT     Yel
74    LD      EMG
      OUT     Red
      ANI     M200  ; Off Buzer
      OUT     Buzzer
END_FUNCTION_BLOCK

FUNCTION_BLOCK C_ShellCage
VAR_INPUT
  AM : BOOL;
  EMG : BOOL;
  I_M_U_DT : BOOL;
  I_M_D_DT : BOOL;
  I_M_Kep : BOOL;
  I_M_Nha : BOOL;
  I_M_Do_Org : BOOL;
  I_M_Do_Lap : BOOL;
  I_M_U_S : BOOL;
  I_M_D_S : BOOL;
  I_M_U_Jig : BOOL;
  I_M_D_Jig : BOOL;
END_VAR
VAR_OUTPUT
  U_Cyl_DT : BOOL;
  D_Cyl_DT : BOOL;
  Kep : BOOL;
  Nha : BOOL;
  Stopper_Up : BOOL;
  Stopper_Down : BOOL;
  Cyl_U_Jig : BOOL;
  Cyl_D_Jig : BOOL;
  Cyl_U_DT_J : BOOL;
  Cyl_D_DT_J : BOOL;
END_VAR
VAR
  M_U_DT : BOOL;
  A_U_DT : BOOL;
  M_D_DT : BOOL;
  A_D_DT : BOOL;
  M_S_Cyl_DT : INT;
  M_Kep : BOOL;
  A_Kep : BOOL;
  M_Nha : BOOL;
  A_Nha : BOOL;
  M_S_Cyl_Kep : INT;
  M_U_S : BOOL;
  A_U_S : BOOL;
  M_D_S : BOOL;
  A_D_S : BOOL;
  M_S_Stp : INT;
  M_U_Jig : BOOL;
  A_U_Jig : BOOL;
  M_D_Jig : BOOL;
  A_D_Jig : BOOL;
  M_S_UD_J : INT;
END_VAR
VAR_INPUT
  I_M_U_DT_Jig : BOOL;
  I_M_D_DT_Jig : BOOL;
END_VAR
VAR
  M_U_DT_J : BOOL;
  A_U_DT_J : BOOL;
  M_D_DT_J : BOOL;
  A_D_DT_J : BOOL;
  M_S_DT_J : INT;
END_VAR
VAR_INPUT
  A_S_Cyl_Kep : INT;
  A_S_Cyl_DT : INT;
  A_S_Stp : INT;
  A_S_UD_J : INT;
  A_S_DT_J : INT;
  ORG : BOOL;
END_VAR
VAR_OUTPUT
  S_Org : BOOL;
END_VAR
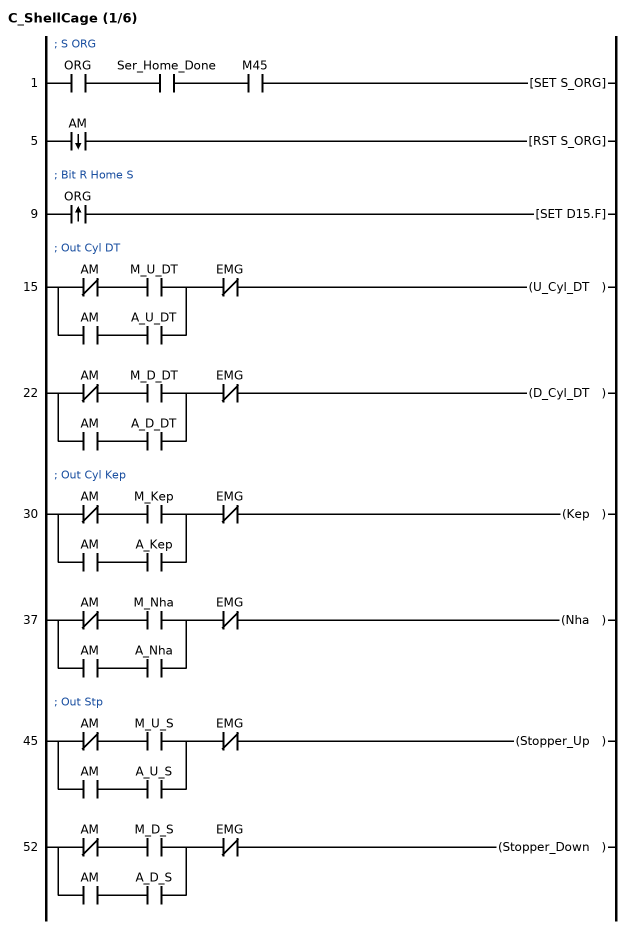
; S ORG
1     LD      ORG
      AND     Ser_Home_Done
      AND     M45
      SET     S_ORG
5     LDF     AM
      RST     S_ORG
; Bit R Home S
9     LDP     ORG
      SET     D15.F
; Out Cyl DT
15    LDI     AM
      AND     M_U_DT
      LD      AM
      AND     A_U_DT
      ORB
      ANI     EMG
      OUT     U_Cyl_DT
22    LDI     AM
      AND     M_D_DT
      LD      AM
      AND     A_D_DT
      ORB
      ANI     EMG
      OUT     D_Cyl_DT
; Out Cyl Kep
30    LDI     AM
      AND     M_Kep
      LD      AM
      AND     A_Kep
      ORB
      ANI     EMG
      OUT     Kep
37    LDI     AM
      AND     M_Nha
      LD      AM
      AND     A_Nha
      ORB
      ANI     EMG
      OUT     Nha
; Out Stp
45    LDI     AM
      AND     M_U_S
      LD      AM
      AND     A_U_S
      ORB
      ANI     EMG
      OUT     Stopper_Up
52    LDI     AM
      AND     M_D_S
      LD      AM
      AND     A_D_S
      ORB
      ANI     EMG
      OUT     Stopper_Down
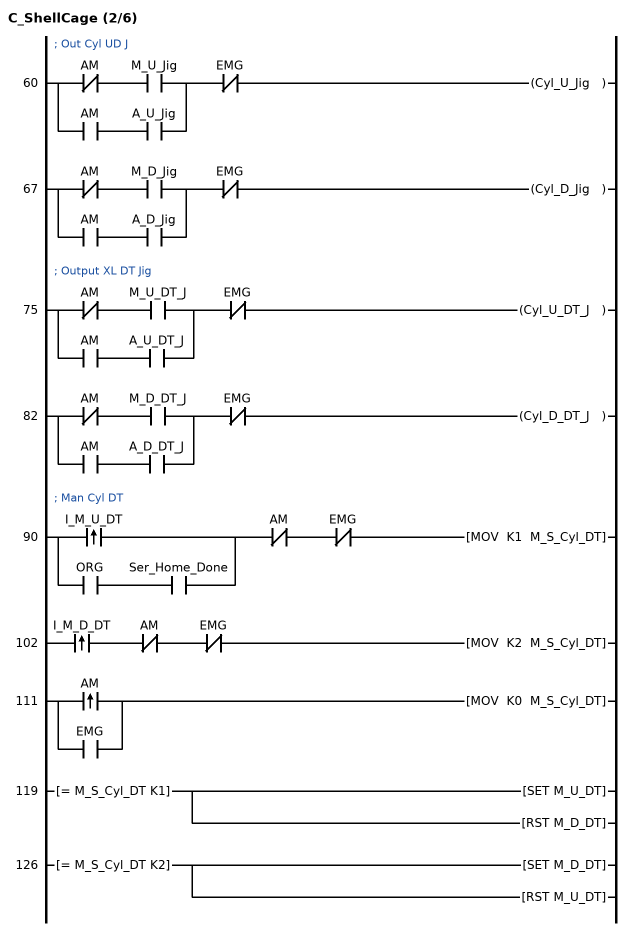
; Out Cyl UD J
60    LDI     AM
      AND     M_U_Jig
      LD      AM
      AND     A_U_Jig
      ORB
      ANI     EMG
      OUT     Cyl_U_Jig
67    LDI     AM
      AND     M_D_Jig
      LD      AM
      AND     A_D_Jig
      ORB
      ANI     EMG
      OUT     Cyl_D_Jig
; Output XL DT Jig
75    LDI     AM
      AND     M_U_DT_J
      LD      AM
      AND     A_U_DT_J
      ORB
      ANI     EMG
      OUT     Cyl_U_DT_J
82    LDI     AM
      AND     M_D_DT_J
      LD      AM
      AND     A_D_DT_J
      ORB
      ANI     EMG
      OUT     Cyl_D_DT_J
; Man Cyl DT
90    LDP     I_M_U_DT
      LD      ORG
      AND     Ser_Home_Done
      ORB
      ANI     AM
      ANI     EMG
      MOV     K1 M_S_Cyl_DT
102   LDP     I_M_D_DT
      ANI     AM
      ANI     EMG
      MOV     K2 M_S_Cyl_DT
111   LDP     AM
      OR      EMG
      MOV     K0 M_S_Cyl_DT
119   LD=     M_S_Cyl_DT K1
      SET     M_U_DT
      RST     M_D_DT
126   LD=     M_S_Cyl_DT K2
      SET     M_D_DT
      RST     M_U_DT
